TEXTLIST CoverConfigTabsTextList
  0 = 'General'
  1 = 'Top'
  2 = 'Bottom'
  3 = 'Top panel 1'
  4 = 'Top panel 2'
  5 = 'Top panel 3'
  6 = 'Top panel 4'
  7 = 'Bottom panel 1'
  8 = 'Bottom panel 2'
  9 = 'Bottom panel 3'
  10 = 'Bottom panel 4'
   = ''
END_TEXTLIST

(* stored: Version 1.1.0.1, ProductVersion 3.1.4018.2
   TextList CoverConfigTabsTextList: Id {f2d28b4f-d88a-4504-bf84-058e4e4d2058} *)
